FUNCTION_BLOCK T_ModuleCollectionAllInAskedStateReturnsCorrectResponse EXTENDS T_UnitTestBase
VAR
  list : T_SubModuleCollection;
  newModule, newModule2 : T_SubModuleMock; 
  actual1, actual2 : BOOL;
END_VAR

// Arrange
list.AddModule(newModule);
list.AddModule(newModule2);

//Act
newModule._Currentstate := Tc3_PackML_V2.E_PMLState.ePMLState_Completing;
newModule2._Currentstate := Tc3_PackML_V2.E_PMLState.ePMLState_Completing;

//Assert
actual1 := list.AllInAskedState(Tc3_PackML_V2.E_PMLState.ePMLState_Completing);

assertion.AssertEquals_BOOL(TRUE, actual1, 'actual1 := list.AllInAskedState(Tc3_PackML_V2.E_PMLState.ePMLState_Completing');
TestFinished();

END_FUNCTION_BLOCK

(* stored: Version 1.1.0.1, ProductVersion 3.1.4024.12
   POU T_ModuleCollectionAllInAskedStateReturnsCorrectResponse: Id {4d3bed85-2a38-44a7-b6fa-f503b71f4f97}, SpecialFunc None *)
